// Mitsubishi GX Works2 project: a5   PLC: Q02/Q02H

PROGRAM MAIN
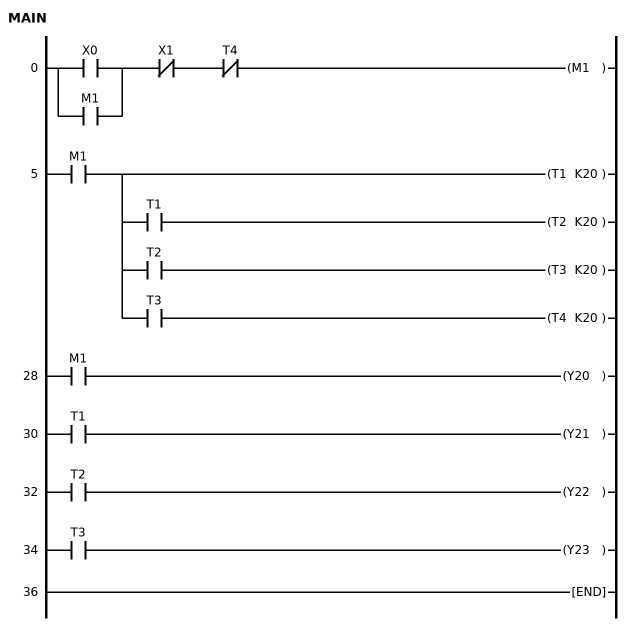
0     LD      X0
      OR      M1
      ANI     X1
      ANI     T4
      OUT     M1
5     LD      M1
      OUT     T1 K20
      MPS
      AND     T1
      OUT     T2 K20
      MRD
      AND     T2
      OUT     T3 K20
      MPP
      AND     T3
      OUT     T4 K20
28    LD      M1
      OUT     Y20
30    LD      T1
      OUT     Y21
32    LD      T2
      OUT     Y22
34    LD      T3
      OUT     Y23
36    END
END_PROGRAM
